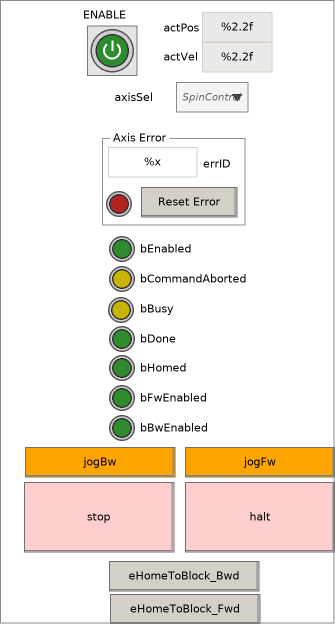
VISUALIZATION StepBlockDetection  // 335x624
    GroupBox (102,130 143x95), "Axis Error"
    Lamp1 (104,189 30x30), variable: GVL.astAxes[MAIN.hmiAxisSelection].stStatus.bError, style: Lamp-Lamp1-Red
    Button (141,187 96x30), "Reset Error", pressed state: GVL.astAxes[MAIN.hmiAxisSelection].stControl.bReset, text list: 'languageTable', text index: "reset"
        OnMouseClick: toggle GVL.astAxes[MAIN.hmiAxisSelection].stControl.bReset
    Textfield (108,147 89x30), "%x", text variable: GVL.astAxes[MAIN.hmiAxisSelection].stStatus.nErrorID
    Textfield (200,149 44x30), "errID", text list: 'languageTable', text index: "errID"
    Textfield (137,413 117x30), "bBwEnabled", text list: 'languageTable', text index: "bBwEnabled"
    Lamp1 (107,234 30x30), variable: GVL.astAxes[MAIN.hmiAxisSelection].stStatus.bEnabled, style: Lamp-Lamp1-Green
    Textfield (137,234 117x30), "bEnabled", text list: 'languageTable', text index: "bEnabled"
    Lamp1 (107,264 30x30), variable: GVL.astAxes[MAIN.hmiAxisSelection].stStatus.bCommandAborted, style: Lamp-Lamp1-Yellow
    Textfield (137,264 117x30), "bCommandAborted", text list: 'languageTable', text index: "bCommandAborted"
    Textfield (137,294 117x30), "bBusy", text list: 'languageTable', text index: "bBusy"
    Lamp1 (107,324 30x30), variable: GVL.astAxes[MAIN.hmiAxisSelection].stStatus.bDone, style: Lamp-Lamp1-Green
    Textfield (137,324 117x30), "bDone", text list: 'languageTable', text index: "bDone"
    Lamp1 (107,353 30x30), variable: GVL.astAxes[MAIN.hmiAxisSelection].stStatus.bHomed, style: Lamp-Lamp1-Green
    Textfield (137,353 117x30), "bHomed", text list: 'languageTable', text index: "bHomed"
    Lamp1 (107,383 30x30), variable: GVL.astAxes[MAIN.hmiAxisSelection].stStatus.bFwEnabled AND NOT GVL.astAxes[MAIN.hmiAxisSelection].stStatus.bInterlockedFwd, style: Lamp-Lamp1-Green
    Lamp1 (107,413 30x30), variable: GVL.astAxes[MAIN.hmiAxisSelection].stStatus.bBwEnabled AND NOT GVL.astAxes[MAIN.hmiAxisSelection].stStatus.bInterlockedBwd, style: Lamp-Lamp1-Green
    Textfield (137,383 117x30), "bFwEnabled", text list: 'languageTable', text index: "bFwEnabled"
    Lamp1 (106,295 30x30), variable: GVL.astAxes[MAIN.hmiAxisSelection].stStatus.bBusy, style: Lamp-Lamp1-Yellow
    Textfield (202,12 70x30), "%2.2f", text variable: GVL.astAxes[MAIN.hmiAxisSelection].stStatus.fActPosition
    Textfield (148,13 54x30), "actPos", text list: 'languageTable', text index: "actposition"
    Textfield (152,42 49x30), "actVel", text list: 'languageTable', text index: "actVelocity"
    Textfield (202,42 70x30), "%2.2f", text variable: GVL.astAxes[MAIN.hmiAxisSelection].stStatus.fActVelocity
    Textfield (80,2 92x26), "ENABLE", text list: 'languageSupport', text index: "enable"
    PowerSwitch (87,24 50x53), variable: GVL.astAxes[MAIN.hmiAxisSelection].stControl.bEnable, behaviour: TOGGLE, style: Switch-PowerSwitch-Green
    Button (25,447 150x30), "jogBw", text list: "languageSupport", text index: "jogBw"
        OnMouseDown: execute { GVL.astAxes[MAIN.hmiAxisSelection].stControl.eCommand:=E_MotionFunctions.eJog; GVL.astAxes[MAIN.hmiAxisSelection].stControl.bJogBwd:= TRUE; }
        OnMouseClick: execute {  }
        OnMouseUp: execute { GVL.astAxes[MAIN.hmiAxisSelection].stControl.bJogBwd:= FALSE; }
    Button (185,447 150x30), "jogFw", text list: "languageSupport", text index: "jogFw"
        OnMouseDown: execute { GVL.astAxes[MAIN.hmiAxisSelection].stControl.eCommand:=E_MotionFunctions.eJog; GVL.astAxes[MAIN.hmiAxisSelection].stControl.bJogFwd:= TRUE; }
        OnMouseClick: execute {  }
        OnMouseUp: execute { GVL.astAxes[1].stControl.bJogFwd:= FALSE; }
    Button (185,482 150x70), "halt", pressed state: GVL.astAxes[1].stControl.bHalt, input disabled if: GVL.astAxes[1].stStatus.bGeared, text list: "languageSupport", text index: "halt"
        toggle GVL.astAxes[MAIN.hmiAxisSelection].stControl.bHalt
    Button (24,482 150x70), "stop", pressed state: GVL.astAxes[1].stControl.bStop, input disabled if: GVL.astAxes[MAIN.hmiAxisSelection].stStatus.bGeared, text list: "languageSupport", text index: "stop"
        toggle GVL.astAxes[MAIN.hmiAxisSelection].stControl.bStop
    Button (109,561 150x30), "eHomeToBlock_Bwd", input disabled if: GVL.astAxes[MAIN.hmiAxisSelection].stStatus.bGeared
        OnMouseClick: execute {
            GVL.astAxes[MAIN.hmiAxisSelection].stControl.eCommand:=E_MotionFunctions.eHome;
            GVL.astAxes[MAIN.hmiAxisSelection].stConfig.eHomeSeq:=E_HomingRoutines.eHomeToBlock_Bwd;
            GVL.astAxes[MAIN.hmiAxisSelection].stControl.bExecute:=TRUE;
        }
    Button (110,594 150x30), "eHomeToBlock_Fwd", input disabled if: GVL.astAxes[MAIN.hmiAxisSelection].stStatus.bGeared
        OnMouseClick: execute {
            GVL.astAxes[MAIN.hmiAxisSelection].stControl.eCommand:=E_MotionFunctions.eHome;
            GVL.astAxes[MAIN.hmiAxisSelection].stConfig.eHomeSeq:=E_HomingRoutines.eHomeToBlock_Fwd;
            GVL.astAxes[MAIN.hmiAxisSelection].stControl.bExecute:=TRUE;
        }
    Textfield (91,85 86x25), "axisSel", text variable: GVL_APP.nAXIS_NUM, text list: "languageSupport", text index: "axisSel"
    SpinControl (176,82 72x30), variable: MAIN.hmiAxisSelection
        p651134158: GVL_APP.nAXIS_NUM
END_VISUALIZATION

(* stored: Version 1.1.0.1, ProductVersion 3.1.4024.10
   Visu StepBlockDetection: Id {1797c93a-675d-4e62-80f4-c8cc8fe9d099} *)
